TYPE "Ttest"
VERSION : 0.1
   STRUCT
      fp_HP : Bool;
      fp_WP : Bool;
      fp_IDLE : Bool;
      WP_on : Bool;
      HP_DUMMY : Bool;
      WP_DUMMY : Bool;
      IDLE_DUMMY : Bool;
   END_STRUCT;

END_TYPE

